(* CODESYS project CommandPatterExport.export

Project tree, tasks and I/O mapping:
  Commands/
    interface ICommand: Execute
    function block CommandQueue [ST]: Dequeue, Enqueue, IsCommandPending
  Machine/
    function block CleanCommand [ST]: Execute
    function block MachineControl [ST]: Clean, Purge, Run, Stop
    function block PurgeCommand [ST]: Execute
  program PLC_PRG [ST]
*)

// PLC_PRG
PROGRAM PLC_PRG
VAR
	Commands : CommandQueue;
	currentCommand : ICommand;
	canExecute : BOOL;
	isDequeued : BOOL;
	
	// Command objects
	startPump : PurgeCommand;
	stopPump : CleanCommand;	
END_VAR


IF Commands.IsCommandPending  AND canExecute THEN
	isDequeued := Commands.Dequeue(ADR(currentCommand));
END_IF
	
IF isDequeued THEN
	currentCommand.Execute();
	isDequeued := FALSE;
END_IF

END_PROGRAM

// Commands/CommandQueue
FUNCTION_BLOCK PUBLIC CommandQueue
VAR CONSTANT
	MaxSize : BYTE := 10;
END_VAR
VAR
	_head : BYTE;
	_tail : BYTE;
	_count : BYTE;
	_commandBuffer : ARRAY[0..MaxSize -1] OF ICommand;
END_VAR

METHOD PUBLIC Dequeue : BOOL
VAR_INPUT
	command : POINTER TO ICommand;
END_VAR

IF _count > 0 AND command > 0 THEN
    command^ := _commandBuffer[_head];
	_head := (_head + 1) MOD MaxSize;
    _count := _count - 1;
	
	Dequeue := TRUE;
ELSE
	Dequeue := FALSE;
END_IF
END_METHOD

METHOD PUBLIC Enqueue : BOOL
VAR_INPUT
	command : ICommand;
END_VAR

IF _count < MaxSize THEN
    _commandBuffer[_tail] := command;
    _tail := (_tail + 1) MOD MaxSize;
    _count := _count + 1;
	
    Enqueue := TRUE;
ELSE
    Enqueue := FALSE;
END_IF
END_METHOD

PROPERTY PUBLIC IsCommandPending : BOOL
GET

IsCommandPending := _count > 0;
END_GET
END_PROPERTY

END_FUNCTION_BLOCK

// Commands/ICommand
INTERFACE ICommand

METHOD Execute
END_METHOD

END_INTERFACE

// Machine/PurgeCommand
FUNCTION_BLOCK PUBLIC PurgeCommand IMPLEMENTS ICommand
VAR_IN_OUT
	Machine : MachineControl;
END_VAR

METHOD PUBLIC Execute
VAR_INPUT
END_VAR

// Perform some checks
Machine.Run();
END_METHOD

END_FUNCTION_BLOCK

// Machine/MachineControl
FUNCTION_BLOCK PUBLIC MachineControl
VAR_INPUT
END_VAR
VAR_OUTPUT
END_VAR
VAR
END_VAR

METHOD Clean : BOOL
END_METHOD

METHOD Purge : BOOL
VAR_INPUT
END_VAR
END_METHOD

METHOD PUBLIC Run : BOOL
VAR_INPUT
END_VAR
END_METHOD

METHOD Stop : BOOL
VAR_INPUT
END_VAR
END_METHOD

END_FUNCTION_BLOCK

// Machine/CleanCommand
FUNCTION_BLOCK PUBLIC CleanCommand IMPLEMENTS ICommand
VAR_IN_OUT
	Machine : MachineControl;
END_VAR

METHOD PUBLIC Execute
VAR_INPUT
END_VAR

// Perform some pre-checks
Machine.Clean();
END_METHOD

END_FUNCTION_BLOCK
